{attribute 'qualified_only'}
{attribute 'strict'}
{attribute 'to_string'}
TYPE E_MESSAGE_FLOW :
(
  MSG_FLOW_INIT,
  MSG_FLOW_ROOT                 := 10,
  MSG_FLOW_ROOT_CREATE,
  MSG_FLOW_ROOT_CREATE_BUSY,
  MSG_FLOW_FOLDER,
  MSG_FLOW_FOLDER_CREATE,
  MSG_FLOW_FOLDER_CREATE_BUSY,
  MSG_FLOW_FILE_CREATE_DONE,
  MSG_FLOW_LINE_START           := 100,
  MSG_FLOW_LINE_BUILD,
  MSG_FLOW_LINE_CHECK,
  MSG_FLOW_WRITE_FILE_BUSY      := 200,
  MSG_FLOW_WRITE_FILE_END,
  MSG_FLOW_WRITE_FILE_DONE      := 1000
)UINT;
END_TYPE

(* stored: Version 1.1.0.1
   DUT E_MESSAGE_FLOW: Id {dcf149f1-8fe7-4e1b-9217-8dbfde1d4038} *)
